{attribute 'GeneratedUsingTerminal: EP8309-0022-0021'}
{attribute addProperty BoxType "EP8309-0022-0021"}
{attribute addProperty Id "Enable_ditheringBOOL1EnableBOOL1ResetBOOL1"}
{attribute addProperty CRC "625230245"}
{attribute addProperty Size "3"}
TYPE Control_254441A5 :
STRUCT
	{attribute addProperty Name "Enable_dithering"}
	Enable_dithering : BOOL;
	{attribute addProperty Name "Enable"}
	Enable : BOOL;
	{attribute addProperty Name "Reset"}
	Reset : BOOL;
END_STRUCT
END_TYPE

(* stored: Version 1.2.0.0, ProductVersion 3.1.4024.9
   DUT Control_254441A5: Id {7c0da96e-b85b-495f-9d8b-2903ee09a6dc} *)
